SUBAPPLICATION Uebung_233_AX (* 3 Taster (I1/I2/I3) auf 1 SR-Latch (Last-Wins) via 3x AX_ASR_RF_TRIG + ASR_MERGE_3 + ASR_AX_SR, Ausgang Q1 *)
  (* Standard: 61499-2; Description: Copyright (c) 2026 Meisterschulen am Ostbahnhof This program and the accompanying materials are made available under the terms of the Eclipse Public License 2.0 which is available at https://www.eclipse.org/legal/epl-2.0/ SPDX-License-Identifier: EPL-2.0 *)
  (* Version 1.0, 2026-09-07, Franz Höpfinger, Meisterschulen am Ostbahnhof, initial API and implementation and/or initial documentation *)
  PACKAGE Uebungen;
  IMPORT logiBUS::io::DI::logiBUS_DI::Input_I1;
  IMPORT logiBUS::io::DI::logiBUS_DI::Input_I2;
  IMPORT logiBUS::io::DI::logiBUS_DI::Input_I3;
  IMPORT logiBUS::io::DQ::logiBUS_DO::Output_Q1;
  (* Documentation:
  3 Taster über ASR_MERGE_3 auf 1 gemeinsames Latch
   Fortsetzung von Uebung_230_AX ("2 Taster, Last-Wins" via ASR_MERGE_2): hier sind es drei unabhängige Taster, zusammengeführt über ASR_MERGE_3. Zeigt, dass die MERGE-Familie kein reiner 2-Input-Spezialfall ist, sondern für beliebig viele Quellen existiert (ASR_MERGE_2..7).
   Funktionsbeschreibung
    - Jeder der drei Taster (Input_I1..I3) wird über einen eigenen AX_ASR_RF_TRIG beobachtet: Drücken → SET, Loslassen → RESET, als gebündeltes ASR.
   - ASR_MERGE_3 führt alle drei ASR-Streams zu einem gemeinsamen zusammen - strukturell identisch zu ASR_MERGE_2 in Uebung_230_AX, nur mit einem dritten Socket (IN3).
   - ASR_AX_SR latcht das gemergte Signal wie gehabt: Last-Wins - welcher Taster zuletzt gedrückt ODER losgelassen wurde (egal welcher der drei), bestimmt den Zustand von Q1.
    Arbeitsauftrag
   Testen Sie: jeder der drei Taster kann Q1 beliebig oft in beliebiger Reihenfolge ein- und ausschalten (Last-Wins, wie in 229/230 - siehe dort für die genaue Funktionsbeschreibung des Last-Wins-Verhaltens). Vergleichen Sie mit Uebung_230_AX: identisches Muster, nur eine Quelle mehr.
  *)
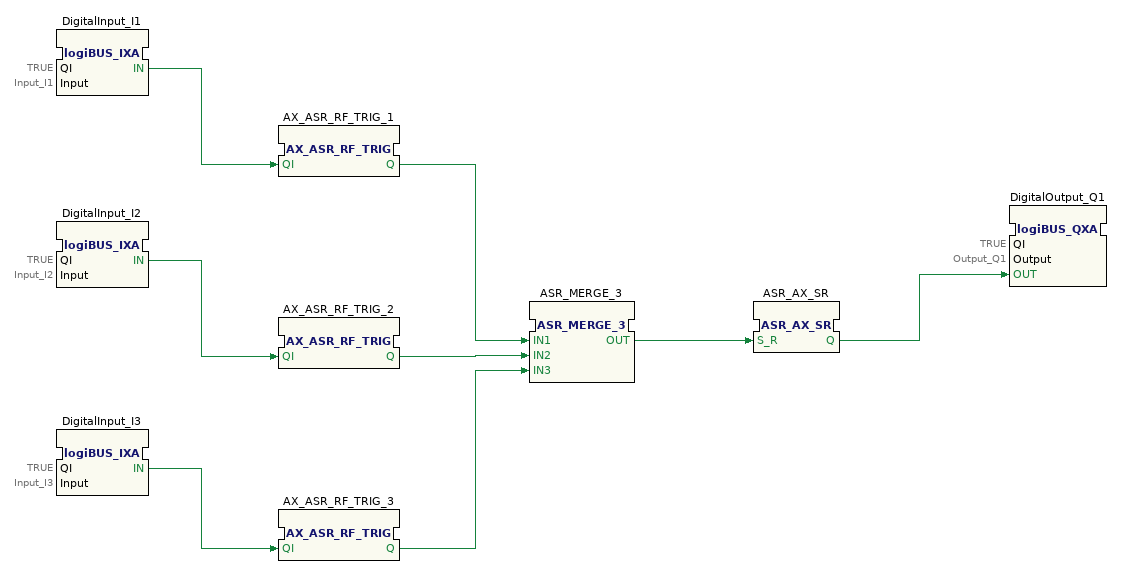
  (* Fortsetzung von Uebung_230_AX: dort fuehrte ASR_MERGE_2 genau 2 Quellen zusammen. Hier zeigt ASR_MERGE_3 mit 3 Quellen, dass die MERGE-Familie kein reiner 2-Input-Spezialfall ist - dieselbe ODER-Verknuepfung, nur mit einem IN3 mehr. *)
  FBS
    DigitalInput_I1 : logiBUS::io::DI::logiBUS_IXA(QI := TRUE, Input := Input_I1);
    DigitalInput_I2 : logiBUS::io::DI::logiBUS_IXA(QI := TRUE, Input := Input_I2);
    DigitalInput_I3 : logiBUS::io::DI::logiBUS_IXA(QI := TRUE, Input := Input_I3);
    AX_ASR_RF_TRIG_1 : adapter::events::unidirectional::AX_ASR_RF_TRIG;
    AX_ASR_RF_TRIG_2 : adapter::events::unidirectional::AX_ASR_RF_TRIG;
    AX_ASR_RF_TRIG_3 : adapter::events::unidirectional::AX_ASR_RF_TRIG;
    ASR_MERGE_3 : adapter::events::unidirectional::ASR_MERGE_3;
    ASR_AX_SR : adapter::events::unidirectional::ASR_AX_SR;
    DigitalOutput_Q1 : logiBUS::io::DQ::logiBUS_QXA(QI := TRUE, Output := Output_Q1);
  END_FBS
  ADAPTER_CONNECTIONS
    DigitalInput_I1.IN TO AX_ASR_RF_TRIG_1.QI;
    DigitalInput_I2.IN TO AX_ASR_RF_TRIG_2.QI;
    DigitalInput_I3.IN TO AX_ASR_RF_TRIG_3.QI;
    AX_ASR_RF_TRIG_1.Q TO ASR_MERGE_3.IN1;
    AX_ASR_RF_TRIG_2.Q TO ASR_MERGE_3.IN2;
    AX_ASR_RF_TRIG_3.Q TO ASR_MERGE_3.IN3;
    ASR_MERGE_3.OUT TO ASR_AX_SR.S_R;
    ASR_AX_SR.Q TO DigitalOutput_Q1.OUT;
  END_CONNECTIONS
END_SUBAPPLICATION
